FUNCTION_BLOCK fb_eventListGenerator
VAR_INPUT
	in_flg_run : BOOL;
	in_var_alarmLevel : eP_alarmLevel;
	in_var_alarmName : WSTRING;
	in_var_alarmMassge : WSTRING;
	in_var_alarmTime : DT;
	in_var_alarmCode1 : eP_alarmCode;
	in_var_alarmCode2 : UDINT;
END_VAR
VAR_IN_OUT
	var_semaphore : INT;
	var_alarmQty : INT;
	var_alarmListLog: s_alarmList;
	out_var_alarmListActive:ARRAY[1..10] OF s_str_alarmList;
END_VAR
VAR_OUTPUT
	out_flg_request : BOOL;
END_VAR
VAR
	buf_var_alarmList : s_alarmList;
	buf_var_str_alarmList : s_str_alarmList;
	flg_active: BOOL;
	buf_var_semaphore: INT;
	var_process: INT;

	delayTimer: TON;
END_VAR

VAR_STAT
	flg_LvError : BOOL;
	flg_LvWarning : BOOL;
	flg_LvInfo : BOOL;
END_VAR
VAR // added by the converter: edge detectors and wires of the graphical bodies
    _rt1, _rt2, _rt3, _rt4 : R_TRIG;
    _w1, _w2, _w3, _w4, _w5 : BOOL;
    _ft1, _ft2 : F_TRIG;
END_VAR

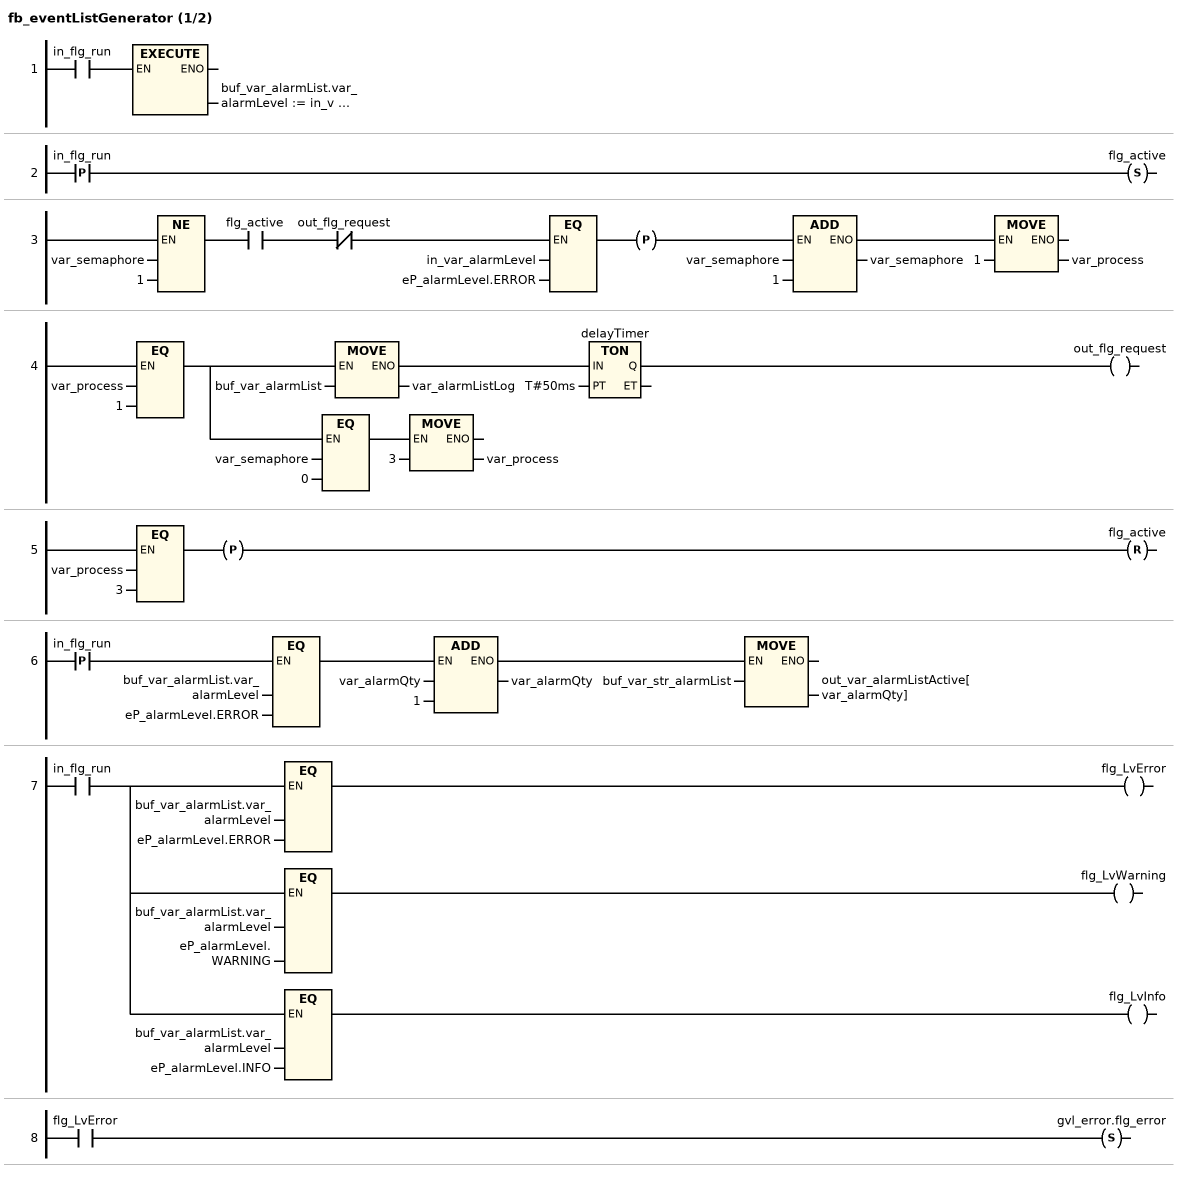
// NETWORK 1
IF in_flg_run THEN
    buf_var_alarmList.var_alarmLevel := in_var_alarmLevel;
    buf_var_alarmList.var_alarmName := in_var_alarmName;
    buf_var_alarmList.var_alarmMassge := in_var_alarmMassge;
    buf_var_alarmList.var_alarmTime := in_var_alarmTime;
    buf_var_alarmList.var_alarmCode1 := in_var_alarmCode1;
    buf_var_alarmList.var_alarmCode2 := in_var_alarmCode2;
    
    
    buf_var_str_alarmList.var_alarmName := in_var_alarmName;
    buf_var_str_alarmList.var_alarmMassge := in_var_alarmMassge;
    buf_var_str_alarmList.var_alarmTime := DT_TO_STRING(in_var_alarmTime);
    buf_var_str_alarmList.var_alarmCode1 := in_var_alarmCode1;
    buf_var_str_alarmList.var_alarmCode2 := UDINT_TO_STRING(in_var_alarmCode2);
END_IF

// NETWORK 2
_rt1(CLK := in_flg_run);
flg_active S= _rt1.Q;

// NETWORK 3
_rt2(CLK := var_semaphore <> 1 AND flg_active AND NOT out_flg_request AND in_var_alarmLevel = eP_alarmLevel.ERROR);
_w1 := _rt2.Q;
IF _w1 THEN var_semaphore := var_semaphore + 1; END_IF
IF _w1 THEN var_process := 1; END_IF

// NETWORK 4
_w2 := var_process = 1;
IF _w2 THEN var_alarmListLog := buf_var_alarmList; END_IF
delayTimer(IN := _w2, PT := T#50ms); // TON
out_flg_request := delayTimer.Q;
IF _w2 AND var_semaphore = 0 THEN var_process := 3; END_IF

// NETWORK 5
_rt3(CLK := var_process = 3);
flg_active R= _rt3.Q;

// NETWORK 6
_rt4(CLK := in_flg_run);
_w3 := _rt4.Q AND buf_var_alarmList.var_alarmLevel = eP_alarmLevel.ERROR;
IF _w3 THEN var_alarmQty := var_alarmQty + 1; END_IF
IF _w3 THEN out_var_alarmListActive[var_alarmQty] := buf_var_str_alarmList; END_IF

// NETWORK 7
flg_LvError := in_flg_run AND buf_var_alarmList.var_alarmLevel = eP_alarmLevel.ERROR;
flg_LvWarning := in_flg_run AND buf_var_alarmList.var_alarmLevel = eP_alarmLevel.WARNING;
flg_LvInfo := in_flg_run AND buf_var_alarmList.var_alarmLevel = eP_alarmLevel.INFO;

// NETWORK 8
gvl_error.flg_error S= flg_LvError;

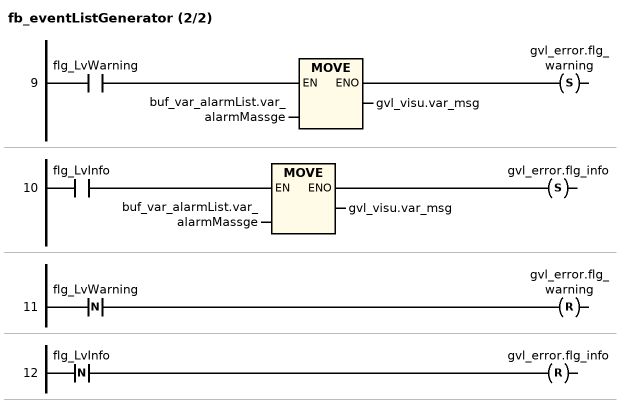
// NETWORK 9
_w4 := flg_LvWarning;
IF _w4 THEN gvl_visu.var_msg := buf_var_alarmList.var_alarmMassge; END_IF
gvl_error.flg_warning S= _w4;

// NETWORK 10
_w5 := flg_LvInfo;
IF _w5 THEN gvl_visu.var_msg := buf_var_alarmList.var_alarmMassge; END_IF
gvl_error.flg_info S= _w5;

// NETWORK 11
_ft1(CLK := flg_LvWarning);
gvl_error.flg_warning R= _ft1.Q;

// NETWORK 12
_ft2(CLK := flg_LvInfo);
gvl_error.flg_info R= _ft2.Q;

END_FUNCTION_BLOCK

(* stored: Version 1.1.0.1, ProductVersion 3.1.4024.11
   POU fb_eventListGenerator: Id {1255accf-829d-4a00-aba7-cdeb275e1ba8}, SpecialFunc None *)
